# B&R Automation Studio project DriveControl1
Automation Studio 4.5.2.102; Default project

## Configuration SampleText

CPU 4PP065.0571-P74, AutomationRuntime D4.52, Build 4.1.2, Vc V4.25.0, Safety 1.6

### Hardware
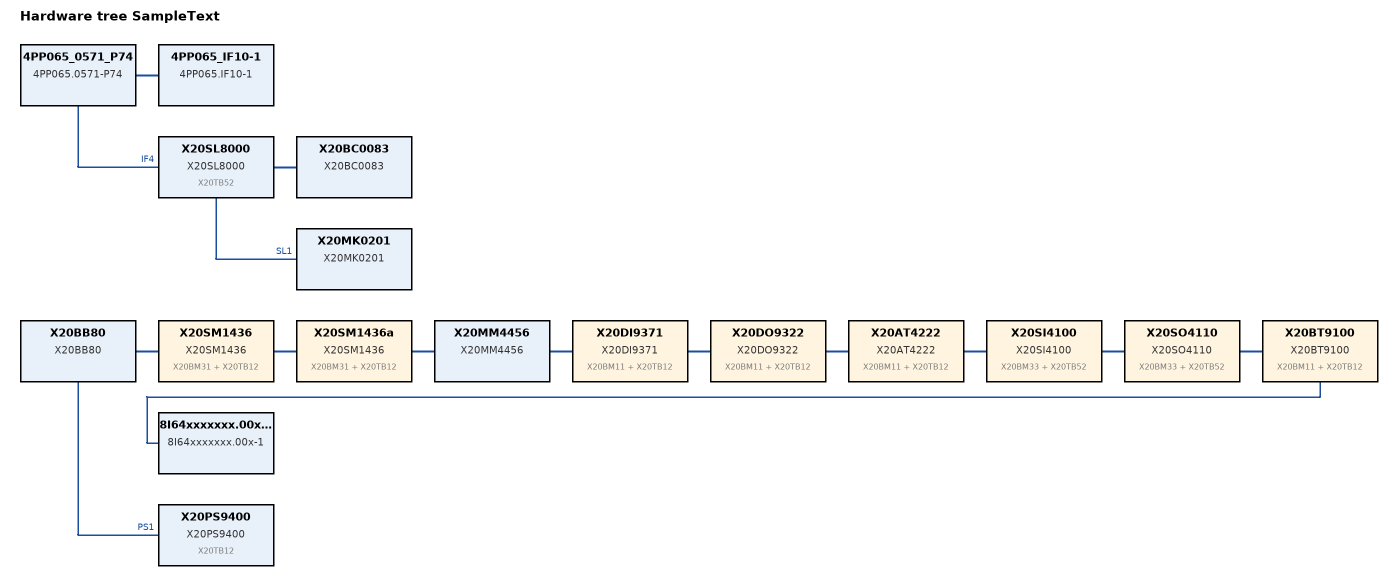
```
4PP065_0571_P74 : 4PP065.0571-P74 v1.1.2.0
  Connector IF5:
    ActivateDevice = 1
    Mode = Manual
    InternetAddress = 10.0.1.10
    SubnetMask = 255.255.255.0
  ConfigurationID = labBR
  TimerDeviceType = EPLX2X
  TimerDevice = 4PP065_0571_P74.IF4
  TaskClassIdleTime = 2000
  Cyclic1Duration = 2000
  Cyclic1Tolerance = 0
  Cyclic1Output = 1
4PP065_IF10-1 : 4PP065.IF10-1 v1.0.3.0  [SS -> 4PP065_0571_P74.SS1]
8I64xxxxxxx.00x-1 : 8I64xxxxxxx.00x-1 v1.3.9.1  [X2X1 -> X20BT9100.X2X1 [Cable Type=X2XCable, Length=10, Version=1.0.0.2]]
  FunctionModel = Standard
  packedETAD = packed
  packedCMDD = packed
  UNS = 220
  NCR = 10
  NSP = 890
  COS = 64
  RSC = 33000
X20AT4222 : X20AT4222 v1.2.3.0  [SS1 -> X20TB12e.SS; SL -> X20BM11c.SL1]
X20BB80 : X20BB80 v1.0.2.0
X20BC0083 : X20BC0083 v2.7.0.0  [PLK1 -> X20SL8000.PLK2 (NodeNumber=2) [Cable Type=PowerlinkCable, Length=10, Version=1.0.0.2]; SL -> X20BB80.SL1]
X20BM11 : X20BM11 v1.0.0.1  [X2X1 -> X20BM33a.X2X2]
X20BM11a : X20BM11 v1.0.0.1  [X2X1 -> X20MM4456.X2X2]
X20BM11b : X20BM11 v1.0.0.1  [X2X1 -> X20BM11a.X2X2]
X20BM11c : X20BM11 v1.0.0.1  [X2X1 -> X20BM11b.X2X2]
X20BM31 : X20BM31 v1.0.0.1  [X2X1 -> X20BB80.IF1]
X20BM31a : X20BM31 v1.0.0.1  [X2X1 -> X20BM31.X2X2]
X20BM33 : X20BM33 v1.0.0.4  [X2X1 -> X20BM11c.X2X2]
X20BM33a : X20BM33 v1.0.0.4  [X2X1 -> X20BM33.X2X2]
X20BT9100 : X20BT9100 v1.0.3.0  [SS1 -> X20TB12f.SS; SL -> X20BM11.SL1]
X20DI9371 : X20DI9371 v1.0.2.0  [SS1 -> X20TB12c.SS; SL -> X20BM11a.SL1]
X20DO9322 : X20DO9322 v1.0.3.0  [SS1 -> X20TB12d.SS; SL -> X20BM11b.SL1]
X20MK0201 : X20MK0201 v1.0.0.0  [SL -> X20SL8000.SL1]
X20MM4456 : X20MM4456 v1.1.5.0  [X2X1 -> X20BM31a.X2X2]
X20PS9400 : X20PS9400 v1.0.2.4  [SS1 -> X20TB12.SS; PS -> X20BB80.PS1]
X20SI4100 : X20SI4100 v1.10.1.1  [SS1 -> X20TB52.SS; SL -> X20BM33.SL1]
X20SL8000 : X20SL8000 v1.6.5.1  [PLK1 -> 4PP065_0571_P74.IF4 (NodeNumber=1) [Cable Type=PowerlinkCable, Length=10, Version=1.0.0.2]; PLK2 -> X20BC0083.PLK1 (NodeNumber=1) [Cable Type=PowerlinkCable, Length=10, Version=1.0.0.2]; SS1 -> X20TB52b.SS]
  SafeProject = SafeLOGIC-1
X20SM1436 : X20SM1436 v1.4.2.1  [SS1 -> X20TB12a.SS; SL -> X20BM31.SL1]
X20SM1436a : X20SM1436 v1.4.2.1  [SS1 -> X20TB12b.SS; SL -> X20BM31a.SL1]
X20SO4110 : X20SO4110 v1.10.1.1  [SS1 -> X20TB52a.SS; SL -> X20BM33a.SL1]
  SafeModuleID = 3
X20TB12 : X20TB12 v1.0.0.0
X20TB12a : X20TB12 v1.0.0.0
X20TB12b : X20TB12 v1.0.0.0
X20TB12c : X20TB12 v1.0.0.0
X20TB12d : X20TB12 v1.0.0.0
X20TB12e : X20TB12 v1.0.0.0
X20TB12f : X20TB12 v1.0.0.0
X20TB52 : X20TB52 v1.0.0.1
X20TB52a : X20TB52 v1.0.0.1
X20TB52b : X20TB52 v1.0.0.1
```

### IoMap.iom - 4PP065_0571_P74/IoMap.iom
```iecst
VAR_CONFIG
	::Program:DriveSM.state AT %IW."8I64xxxxxxx.00x-1".ETAD_Input;
	::Program:DriveSM.command AT %QW."8I64xxxxxxx.00x-1".CMDD_Output;
	::Program:DriveSM.speed AT %QW."8I64xxxxxxx.00x-1".LFRD_Output;
	::Program:DoorSM.sw1 AT %IX."X20DI9371".DigitalInput02;
	::Program:DoorSM.sw2 AT %IX."X20DI9371".DigitalInput03;
	::Program:DoorSM.sw3 AT %IX."X20DI9371".DigitalInput04;
	::Program:DoorSM.sw4 AT %IX."X20DI9371".DigitalInput05;
	::Program:DoorSM.direction AT %IX."X20DI9371".DigitalInput01;
	::Program:LedSM.led4 AT %QX."X20DO9322".DigitalOutput05;
	::Program:LedSM.led3 AT %QX."X20DO9322".DigitalOutput04;
	::Program:LedSM.led2 AT %QX."X20DO9322".DigitalOutput03;
	::Program:LedSM.led1 AT %QX."X20DO9322".DigitalOutput02;
END_VAR
```

## Configuration Simulation

CPU , AutomationRuntime J4.25

### Task classes (Cpu.sw)
```
Libraries: AsIecCon, astime
```

### Hardware
```
PC_any : PC_any v1.1.0.0 (OrderNumber=PC)
```

## Logical view

Binary libraries used (declarations not repeated): RUNTIME, Operator, AsIecCon, astime, sys_lib, asstring

### Library Logical/Libraries/DriveLib (ANSIC)

#### ConStants.var - Exported constants
```iecst
VAR CONSTANT
	CMD_SWITCHED_ON : USINT := 7;
	CMD_DISABLE_VOLTAGE : USINT := 0;
	CMD_ENABLED : USINT := 15;
	CMD_SHUTDOWN : USINT := 6;
	STATE_READY : USINT := 33;
	STATE_DISABLED : USINT := 64;
	STATE_SWITCHED_ON : USINT := 35;
	ST_INIT : USINT := 0;
	ST_UNKNOWN : USINT := 1;
	ST_OPEN : USINT := 2;
	ST_CLOSE : USINT := 3;
	ST_ACC_POS : USINT := 4;
	ST_ACC_NEG : USINT := 5;
	ST_POS : USINT := 6;
	ST_NEG : USINT := 7;
	ST_DEC_POS : USINT := 8;
	ST_DEC_NEG : USINT := 9;
END_VAR
```

#### DriveLib.fun - Exported functions and function blocks
```iecst
{REDUND_ERROR} FUNCTION_BLOCK DriveStateMachine (*TODO: Add your comment here*) (*$GROUP=User,$CAT=User,$GROUPICON=User.png,$CATICON=User.png*)
	VAR_INPUT
		state : UINT;
		enable : BOOL;
		speed : INT;
	END_VAR
	VAR_OUTPUT
		command : UINT;
	END_VAR
END_FUNCTION_BLOCK

{REDUND_ERROR} FUNCTION_BLOCK DoorStateMachine (*TODO: Add your comment here*) (*$GROUP=User,$CAT=User,$GROUPICON=User.png,$CATICON=User.png*)
	VAR_INPUT
		sw1 : {REDUND_UNREPLICABLE} BOOL;
		sw2 : {REDUND_UNREPLICABLE} BOOL;
		sw3 : {REDUND_UNREPLICABLE} BOOL;
		sw4 : {REDUND_UNREPLICABLE} BOOL;
		direction : {REDUND_UNREPLICABLE} BOOL;
	END_VAR
	VAR_OUTPUT
		speed : {REDUND_UNREPLICABLE} INT;
		state : UINT;
	END_VAR
	VAR
		osw1 : BOOL;
		osw2 : BOOL;
		osw3 : BOOL;
		osw4 : BOOL;
	END_VAR
END_FUNCTION_BLOCK

{REDUND_ERROR} FUNCTION_BLOCK LedStateMachine (*TODO: Add your comment here*) (*$GROUP=User,$CAT=User,$GROUPICON=User.png,$CATICON=User.png*)
	VAR_INPUT
		state : {REDUND_UNREPLICABLE} UINT;
	END_VAR
	VAR_OUTPUT
		led1 : {REDUND_UNREPLICABLE} BOOL;
		led2 : {REDUND_UNREPLICABLE} BOOL;
		led3 : {REDUND_UNREPLICABLE} BOOL;
		led4 : {REDUND_UNREPLICABLE} BOOL;
		timer : {REDUND_UNREPLICABLE} INT := 1;
	END_VAR
END_FUNCTION_BLOCK
```

#### DriveStateMachine.c
```c
#include <bur/plctypes.h>
#ifdef __cplusplus
	extern "C"
	{
#endif
	#include "DriveLib.h"
#ifdef __cplusplus
	};
#endif
/* TODO: Add your comment here */
void DriveStateMachine(struct DriveStateMachine* inst)
{
	UINT mask = inst->state & 0x6f;
	if(!inst->enable)
	{
		inst->command = CMD_SHUTDOWN;
	}
	else
	{
		switch (mask)
		{
			case STATE_DISABLED:
				inst->command = CMD_SHUTDOWN;
				break;

			case STATE_READY:
				inst->command = CMD_ENABLED;
				break;

			case STATE_SWITCHED_ON:
				inst->command = CMD_SWITCHED_ON;
				break;
		}
	}
}
```

#### DoorStateMachine.c
```c
#include <bur/plctypes.h>
#ifdef __cplusplus
	extern "C"
	{
#endif
	#include "DriveLib.h"
#ifdef __cplusplus
	};
#endif
/* TODO: Add your comment here */
void DoorStateMachine(struct DoorStateMachine* inst)
{
	inst->direction=!inst->direction;

	//State init
	/*if(inst->sw1==0 && inst->sw2==0 && inst->sw3==0 && inst->sw4==0)
	{
		inst->state = ST_INIT;
	}
	if(inst->state == ST_INIT)
	{

		inst->state = ST_UNKNOWN;
	}
	//state unknown
	if(inst->state == ST_UNKNOWN)
	{
		inst->state = ST_CLOSE ;
	}*/

	//открытие двери
	if(/*inst->state == ST_CLOSE &&*/ inst->sw1 != inst->osw1 && inst->direction==0)
	{
		inst->state = ST_ACC_POS ;
		inst->speed = -200;
	}

	if(/*inst->state == ST_ACC_POS &&*/ inst->sw2 != inst->osw2 && inst->direction == 0)
	{
		inst->state = ST_POS ;
		inst->speed = -600;
	}

	if(/*inst->state == ST_POS  &&*/ inst->sw3 != inst->osw3 && inst->direction == 0)
	{
		inst->state = ST_DEC_POS;
		inst->speed = -200;
	}

	if(/*inst->state == ST_DEC_POS &&*/ inst->sw4 != inst->osw4 && inst->direction == 0)
	{
		inst->state = ST_OPEN;
		inst->speed = 0;
	}

	//закрытие двери
	if(/*inst->state == ST_OPEN &&*/ inst->sw4 != inst->osw4 && inst->direction==1)
	{
		inst->state = ST_ACC_NEG;
		inst->speed = 200;
	}

	if(/*inst->state == ST_ACC_NEG &&*/ inst->sw3 != inst->osw3 && inst->direction == 1)
	{
		inst->state = ST_NEG;
		inst->speed = 600;
	}

	if(/*inst->state == ST_NEG &&*/ inst->sw2 != inst->osw2 && inst->direction == 1)
	{
		inst->state = ST_DEC_NEG;
		inst->speed = 200;
	}

	if(/*inst->state == ST_DEC_NEG &&*/ inst->sw1 != inst->osw1 && inst->direction == 1)
	{
		inst->state = ST_CLOSE;
		inst->speed = 0;
	}
	inst->osw1 = inst->sw1;
	inst->osw2 = inst->sw2;
	inst->osw3 = inst->sw3;
	inst->osw4 = inst->sw4;

}
```

#### LedStateMachine.c
```c
#include <bur/plctypes.h>
#ifdef __cplusplus
	extern "C"
	{
#endif
	#include "DriveLib.h"
#ifdef __cplusplus
	};
#endif
/* TODO: Add your comment here */
void LedStateMachine(struct LedStateMachine* inst)
{

	if(inst->state == ST_ACC_POS)
	{
		inst->led1 = 0;
		if(inst->timer == 3 )
		{
			inst->led2 = !inst->led2;
		}
		inst->led3 = 1;
		inst->led4 = 1;
	}

	if(inst->state == ST_POS)
	{
		inst->led1 = 0;
		inst->led2 = 0;
		inst->led3 = !inst->led3;
		inst->led4 = 1;
	}

	if(inst->state == ST_DEC_POS)
	{

		inst->led1 = 0;
		inst->led2 = 0;
		inst->led3 = 0;
		if(inst->timer == 3 )
		{
			inst->led4 = !inst->led4;
		}
	}

	if(inst->state == ST_OPEN)
	{
		inst->led1 = 0;
		inst->led2 = 0;
		inst->led3 = 0;
		inst->led4 = 0;
	}

	//закрытие двери
	if(inst->state == ST_ACC_NEG )
	{
		inst->led1 = 0;
		inst->led2 = 0;
		if(inst->timer == 3 )
		{
			inst->led3 = !inst->led3;
		}
		inst->led4 = 1;
	}

	if(inst->state == ST_NEG)
	{
		inst->led1 = 0;
		inst->led2 =!inst->led2;
		inst->led3 = 1;
		inst->led4 = 1;
	}

	if(inst->state == ST_DEC_NEG )
	{
		if(inst->timer == 3 )
		{
			inst->led1 = !inst->led1;
		}
		inst->led2 = 1;
		inst->led3 = 1;
		inst->led4 = 1;
	}

	if(inst->state == ST_CLOSE)
	{
		inst->led1 = 1;
		inst->led2 = 1;
		inst->led3 = 1;
		inst->led4 = 1;
	}

	if(inst->timer == 3)
		inst->timer = 0;

	inst->timer++;
}
```

### Program Logical/Program (ANSIC)

#### Init.c - Initialization code
```c
#include <bur/plctypes.h>

#ifdef _DEFAULT_INCLUDES
	#include <AsDefault.h>
#endif

void _INIT ProgramInit(void)
{

	DriveSM.enable = 1;
}
```

#### Cyclic.c - Cyclic code
```c
#include <bur/plctypes.h>

#ifdef _DEFAULT_INCLUDES
	#include <AsDefault.h>
#endif

void _CYCLIC ProgramCyclic(void)
{
	DoorStateMachine(&DoorSM);
	DriveSM.speed = DoorSM.speed;
	DriveStateMachine(&DriveSM);
	LedSM.state = DoorSM.state;
	LedStateMachine(&LedSM);
	/*
	DriveSM.speed = 250;
	DriveStateMachine(&DriveSM);
*/
}
```

#### Variables.var - Local variables
```iecst
VAR
	speed : INT := 0;
	DriveSM : DriveStateMachine := (0);
	LedSM : LedStateMachine := (0);
	DoorSM : DoorStateMachine := (0);
END_VAR
```

Listed in the project but not available here: Logical/Libraries/DriveLib/Types.typ, Logical/Program/Exit.c, Logical/Program/Types.typ
